// TIA Portal V18 export
DATA_BLOCK "TEMPLATE--1.0--F_DB"   // DB39, F_DB
{ S7_Optimized_Access := 'TRUE' }
   VAR
      "!ITERATOR_STRINGS$$" : Bool;
   END_VAR
BEGIN
END_DATA_BLOCK
